// SIMATIC STEP 7 (V5.x) project S_M_General
// CPU: CPU312(1)
// station: P_ADR_BUS
// station: Hardware
// station: Equipo SIMATIC 300
// program: Programa S7(1)

SYMBOL_TABLE
"CONTADOR"	C 1	COUNTER
"Global"	DB 1	DB 1
"INFO_BOB"	DB 4	DB 4
"DESBOBINADO"	FB 1	FB 1	// Función que se encarga del desbobinado
"CIZALLADO"	FB 2	FB 2	// Funcion que se encaga del cizallado de planchas
"MULT_DESBOB"	FB 3	FB 3
"MULT_CIZA"	FB 4	FB 4
"MULT_GEN"	FB 5	FB 5
"MULT_GEN_DESB"	FB 6	FB 6
"CORTAR"	FC 1	FC 1	// Funcion de cortar las planchas
"PESAJE"	FC 2	FC 2	// Función de pesaje
"SCALE"	FC 105	FC 105	// Scaling Values
"START"	I 124.0	BOOL
"BIT_DE_TRABAJO"	I 124.1	BOOL
"BOBINA_COLOCADA"	I 124.2	BOOL
"S_SARTEN"	I 124.5	BOOL
"S_CACEROLA"	I 124.6	BOOL
"S_PAELLERA"	I 124.7	BOOL
"S_WOK"	I 125.0	BOOL
"PRESENCIA"	I 125.1	BOOL
"PALET"	I 125.3	BOOL
"SENSORARRIBA"	I 125.4	BOOL
"SENSORABAJO"	I 125.5	BOOL
"EXPULSADA"	I 125.6	BOOL
"PESO_OUT"	MD 100	REAL
"Cycle Execution"	OB 1	OB 1
"MCENTRO"	PIW 651	INT
"IN_PESAJE"	PIW 653	INT
"ABRIRMCENTRO"	Q 100.0	BOOL
"CERRARMCENTRO"	Q 100.1	BOOL
"DESBOBINAR"	Q 100.2	BOOL
"EXPULSAR_BOBINA"	Q 100.3	BOOL
"PRENSA"	Q 100.4	BOOL
"EXPULSAR_PLANCHA"	Q 100.5	BOOL
"BAJAR_CUCHILLA"	Q 100.6	BOOL
"EXPULSAR_PALET"	Q 101.0	BOOL
"STBY"	Q 101.1	BOOL
END_SYMBOL_TABLE

FUNCTION_BLOCK "DESBOBINADO"	// FB 1
TITLE = DESBOBINADO
VERSION : 0.1
VAR_INPUT
  SENSOR : BOOL ;
  PRESENCIA : BOOL ;
  CENTRO : INT ;
  bit_de_trabajo : BOOL ;
  MCENTRO : INT ;
  Contador : COUNTER ;
  START : BOOL ;
  PLANCHAS : WORD  := W#16#100;
END_VAR
VAR_OUTPUT
  ABRIRMCENTRO : BOOL ;
  DESBOBINAR : BOOL ;
  STBY : BOOL ;
END_VAR
VAR
  x31 : BOOL ;
  x32 : BOOL ;
  x33 : BOOL ;
  x34 : BOOL ;
  s1 : BOOL ;
  FP_Bit_Tr : BOOL ;
  x30 : BOOL ;
  FP_PRESENCIA : BOOL ;
  FP_BDT : BOOL ;
  FP_START : BOOL ;
END_VAR
VAR_TEMP
  watchdog_master : BOOL ;
END_VAR
BEGIN
NETWORK
TITLE = Arranque
      SET;
      A     #bit_de_trabajo;
      FP    #FP_BDT;
      S     #x30;
      R     #x31;
      R     #x32;
      R     #x33;
      R     #x34;
      R     #s1;
NETWORK
TITLE = x31 a x32
//Comparacion medida centro con medida nominal del centro para pasar de x31 a x32
      A     #x31;
      A(;
      L     #CENTRO;
      L     #MCENTRO;
      ==R;
      );
      R     #x31;
      S     #x32;
NETWORK
TITLE = x32 a x33
//Presencia detecta que la plancha esta en posicion para empezar el proceso de 
//desbobinado-cizallado
      A     #x32;
      A     #PRESENCIA;
      FP    #FP_PRESENCIA;
      R     #x32;
      S     #x33;
NETWORK
TITLE = x33 a x34
//Detecta que la plancha esta lista para ser cizallada
      A     #x33;
      A     #SENSOR;
      R     #x33;
      S     #x34;
NETWORK
TITLE = x34 a x33
//si el contador no ha acabado
      A     #x34;
      T     LD 1;
      TAK;
      T     LD 5;
      L     #Contador;
      T     LW 9;
      L     LD 5;
      L     LD 1;
      A     C [LW 9];
      AN    #SENSOR;
      R     #x34;
      S     #x33;
NETWORK
TITLE = x34 a s1
//si el contador ha cabado
      A     #x34;
      T     LD 1;
      TAK;
      T     LD 5;
      L     #Contador;
      T     LW 9;
      L     LD 5;
      L     LD 1;
      AN    C [LW 9];
      AN    #SENSOR;
      AN    #PRESENCIA;
      R     #x34;
      S     #x30;
NETWORK
TITLE = Tratamiento de bit de fin
      A     #x30;
      =     #STBY;
NETWORK
TITLE = Abrir centro
      A     #x31;
      =     #ABRIRMCENTRO;
NETWORK
TITLE = Carga del contador y desbobinado en x32
      A     #x32;
      S     #DESBOBINAR;
      L     #PLANCHAS;
      T     LD 1;
      TAK;
      T     LD 5;
      L     #Contador;
      T     LW 9;
      L     LD 5;
      L     LD 1;
      S     C [LW 9];
NETWORK
TITLE = Resta del contador y salida del x33
      A     #x33;
      S     #DESBOBINAR;
NETWORK
TITLE =
      A     #x34;
      R     #DESBOBINAR;
NETWORK
TITLE = De X30 a X31
      A     #START;
      FP    #FP_START;
      A     #x30;
      R     #x30;
      S     #x31;
END_FUNCTION_BLOCK

FUNCTION_BLOCK "CIZALLADO"	// FB 2
TITLE = CIZALLADO
VERSION : 0.1
VAR_INPUT
  bit_de_trabajo : BOOL ;
  SENSOR : BOOL ;
  SENSORABAJO : BOOL ;
  SENSORARRIBA : BOOL ;
  EXPULSADA : BOOL ;
  CONTADOR : COUNTER ;
  START : BOOL ;
END_VAR
VAR_OUTPUT
  BAJARCUCHILLA : BOOL ;
  EXPULSARPLANCHA : BOOL ;
  STBY : BOOL ;
  BIT_OK : BOOL ;
END_VAR
VAR
  X41 : BOOL ;
  M3 : BOOL ;
  X43 : BOOL ;
  FP_BDT : BOOL ;
  FP_START : BOOL ;
  INICORTAR : BOOL ;
  S2 : BOOL ;
  BDT_CORTAR : BOOL ;
  OK_CORTAR : BOOL ;
  STBY_CORTAR : BOOL ;
  CORTADO : BOOL ;
END_VAR
BEGIN
NETWORK
TITLE = Arranque
      A     #bit_de_trabajo;
      FP    #FP_BDT;
      =     #BDT_CORTAR;
      S     #X41;
      R     #M3;
      R     #X43;
      R     #INICORTAR;
      R     #CORTADO;
      R     #BIT_OK;
      R     #S2;
NETWORK
TITLE = De x41 a M3
      A     #X41;
      A     #SENSOR;
      A     #STBY_CORTAR;
      A     #START;
      FP    #FP_START;
      R     #X41;
      S     #M3;
NETWORK
TITLE = De M3 a x43
      A     #M3;
      A     #CORTADO;
      R     #M3;
      S     #X43;
NETWORK
TITLE = de x43 a x41
      A     #X43;
      T     LD 0;
      TAK;
      T     LD 4;
      L     #CONTADOR;
      T     LW 8;
      L     LD 4;
      L     LD 0;
      AN    C [LW 8];
      R     #X43;
      S     #S2;
NETWORK
TITLE = de x43 a X41
      A     #X43;
      T     LD 0;
      TAK;
      T     LD 4;
      L     #CONTADOR;
      T     LW 8;
      L     LD 4;
      L     LD 0;
      A     C [LW 8];
      R     #X43;
      S     #X41;
NETWORK
TITLE = De M3 a x43 con call M3
      CALL  "CORTAR" (
           bit_de_trabajo           := #BDT_CORTAR,
           SENSORABAJO              := #SENSORABAJO,
           SENSORARRIBA             := #SENSORARRIBA,
           EXPULSADA                := #EXPULSADA,
           START                    := #INICORTAR,
           OK                       := #OK_CORTAR,
           BAJARCUCHILLA            := #BAJARCUCHILLA,
           EXPULSARPLANCHA          := #EXPULSARPLANCHA,
           bit_ok                   := #CORTADO,
           STBY                     := #STBY_CORTAR);
NETWORK
TITLE =
      A     #M3;
      A     #CORTADO;
      R     #M3;
      S     #X43;
NETWORK
TITLE =
      A     #M3;
      =     #INICORTAR;
NETWORK
TITLE = Cuenta el numero de planchas cortadas
      A     #X43;
      =     #OK_CORTAR;
      T     LD 0;
      TAK;
      T     LD 4;
      L     #CONTADOR;
      T     LW 8;
      L     LD 4;
      L     LD 0;
      CD    C [LW 8];
NETWORK
TITLE =
      A     #X41;
      =     #STBY;
NETWORK
TITLE =
      A     #S2;
      =     #BIT_OK;
END_FUNCTION_BLOCK

FUNCTION_BLOCK "MULT_DESBOB"	// FB 3
VERSION : 0.1
VAR_INPUT
  S_CACEROLA : BOOL ;
  S_SARTEN : BOOL ;
  S_PAELLERA : BOOL ;
  S_WOK : BOOL ;
  PRESENCIA : BOOL ;
  C_CACEROLA : INT ;
  C_SARTEN : INT ;
  C_WOK : INT ;
  C_PAELLERA : INT ;
  BIT_DE_TRABAJO : BOOL ;
  MCENTRO : INT ;
  CONTADOR : COUNTER ;
  PLANCHAS : WORD ;
  SARTEN : BOOL ;
  CACEROLA : BOOL ;
  WOK : BOOL ;
  PAELLERA : BOOL ;
  START : BOOL ;
END_VAR
VAR_OUTPUT
  ABRIRMCENTRO : BOOL ;
  DESBOBINAR : BOOL ;
  BIT_OK : BOOL ;
  BIT_ERROR : BOOL ;
  STBY : BOOL ;
END_VAR
VAR
  CAC_DESB : FB 1;
  SART_DESB : FB 1;
  WOK_DESB : FB 1;
  PAELL_DESB : FB 1;
  START_SAR : BOOL ;
  START_CAC : BOOL ;
  START_WOK : BOOL ;
  START_PAELL : BOOL ;
  FP_BDT : BOOL ;
  X1 : BOOL ;
  X2 : BOOL ;
  X3 : BOOL ;
  X4 : BOOL ;
  X5 : BOOL ;
  X6 : BOOL ;
  BDT : BOOL ;
  FP_START : BOOL ;
  FLAG_DESB : BOOL ;
  FP_DESBOB : BOOL ;
  F_START : BOOL ;
  STBY_SAR : BOOL ;
  STBY_CAC : BOOL ;
  STBY_WOK : BOOL ;
  STBY_PAELL : BOOL ;
END_VAR
BEGIN
NETWORK
TITLE =
      A     #X2;
      JCN   _008;
      S     #BDT;
      BLD   14;
      =     L 6.0;
      L     DINO;
      T     LW 4;
      CDB;
      OPN   DI [LW 4];
      TAR2  LD 0;
      A     DBX [AR2,P#0.1];
      =     #SART_DESB.SENSOR;
      A     DBX [AR2,P#0.4];
      =     #SART_DESB.PRESENCIA;
      L     DBW [AR2,P#4.0];
      T     #SART_DESB.CENTRO;
      A     DBX [AR2,P#95.3];
      =     #SART_DESB.bit_de_trabajo;
      L     DBW [AR2,P#12.0];
      T     #SART_DESB.MCENTRO;
      L     DBW [AR2,P#14.0];
      T     #SART_DESB.Contador;
      A     DBX [AR2,P#94.0];
      =     #SART_DESB.START;
      L     DBW [AR2,P#16.0];
      T     #SART_DESB.PLANCHAS;
      +AR2  P#40.0;
      UC    "DESBOBINADO";
      LAR2  LD 0;
      A     #SART_DESB.ABRIRMCENTRO;
      =     DBX [AR2,P#20.0];
      A     #SART_DESB.DESBOBINAR;
      =     DBX [AR2,P#20.1];
      A     #SART_DESB.STBY;
      =     DBX [AR2,P#96.0];
      CDB;
      BLD   15;
_008: NOP   0;
NETWORK
TITLE =
      A     #X3;
      JCN   _009;
      S     #BDT;
      BLD   14;
      =     L 6.0;
      L     DINO;
      T     LW 4;
      CDB;
      OPN   DI [LW 4];
      TAR2  LD 0;
      A     DBX [AR2,P#0.0];
      =     #CAC_DESB.SENSOR;
      A     DBX [AR2,P#0.4];
      =     #CAC_DESB.PRESENCIA;
      L     DBW [AR2,P#2.0];
      T     #CAC_DESB.CENTRO;
      A     DBX [AR2,P#95.3];
      =     #CAC_DESB.bit_de_trabajo;
      L     DBW [AR2,P#12.0];
      T     #CAC_DESB.MCENTRO;
      L     DBW [AR2,P#14.0];
      T     #CAC_DESB.Contador;
      A     DBX [AR2,P#94.1];
      =     #CAC_DESB.START;
      L     DBW [AR2,P#16.0];
      T     #CAC_DESB.PLANCHAS;
      +AR2  P#22.0;
      UC    "DESBOBINADO";
      LAR2  LD 0;
      A     #CAC_DESB.ABRIRMCENTRO;
      =     DBX [AR2,P#20.0];
      A     #CAC_DESB.DESBOBINAR;
      =     DBX [AR2,P#20.1];
      A     #CAC_DESB.STBY;
      =     DBX [AR2,P#96.1];
      CDB;
      BLD   15;
_009: NOP   0;
NETWORK
TITLE =
      A     #X4;
      JCN   _010;
      S     #BDT;
      BLD   14;
      =     L 6.0;
      L     DINO;
      T     LW 4;
      CDB;
      OPN   DI [LW 4];
      TAR2  LD 0;
      A     DBX [AR2,P#0.3];
      =     #WOK_DESB.SENSOR;
      A     DBX [AR2,P#0.4];
      =     #WOK_DESB.PRESENCIA;
      L     DBW [AR2,P#6.0];
      T     #WOK_DESB.CENTRO;
      A     DBX [AR2,P#95.3];
      =     #WOK_DESB.bit_de_trabajo;
      L     DBW [AR2,P#12.0];
      T     #WOK_DESB.MCENTRO;
      L     DBW [AR2,P#14.0];
      T     #WOK_DESB.Contador;
      A     DBX [AR2,P#94.2];
      =     #WOK_DESB.START;
      L     DBW [AR2,P#16.0];
      T     #WOK_DESB.PLANCHAS;
      +AR2  P#58.0;
      UC    "DESBOBINADO";
      LAR2  LD 0;
      A     #WOK_DESB.ABRIRMCENTRO;
      =     DBX [AR2,P#20.0];
      A     #WOK_DESB.DESBOBINAR;
      =     DBX [AR2,P#20.1];
      A     #WOK_DESB.STBY;
      =     DBX [AR2,P#96.2];
      CDB;
      BLD   15;
_010: NOP   0;
NETWORK
TITLE =
      A     #X5;
      JCN   _011;
      S     #BDT;
      BLD   14;
      =     L 6.0;
      L     DINO;
      T     LW 4;
      CDB;
      OPN   DI [LW 4];
      TAR2  LD 0;
      A     DBX [AR2,P#0.2];
      =     #PAELL_DESB.SENSOR;
      A     DBX [AR2,P#0.4];
      =     #PAELL_DESB.PRESENCIA;
      L     DBW [AR2,P#8.0];
      T     #PAELL_DESB.CENTRO;
      A     DBX [AR2,P#95.3];
      =     #PAELL_DESB.bit_de_trabajo;
      L     DBW [AR2,P#12.0];
      T     #PAELL_DESB.MCENTRO;
      L     DBW [AR2,P#14.0];
      T     #PAELL_DESB.Contador;
      A     DBX [AR2,P#94.3];
      =     #PAELL_DESB.START;
      L     DBW [AR2,P#16.0];
      T     #PAELL_DESB.PLANCHAS;
      +AR2  P#76.0;
      UC    "DESBOBINADO";
      LAR2  LD 0;
      A     #PAELL_DESB.ABRIRMCENTRO;
      =     DBX [AR2,P#20.0];
      A     #PAELL_DESB.DESBOBINAR;
      =     DBX [AR2,P#20.1];
      A     #PAELL_DESB.STBY;
      =     DBX [AR2,P#96.3];
      CDB;
      BLD   15;
_011: NOP   0;
NETWORK
TITLE =
      A     #X2;
      =     #START_SAR;
NETWORK
TITLE =
      A     #X3;
      =     #START_CAC;
NETWORK
TITLE =
      A     #X4;
      =     #START_WOK;
NETWORK
TITLE =
      A     #X5;
      =     #START_PAELL;
NETWORK
TITLE =
      A     #BIT_DE_TRABAJO;
      FP    #FP_BDT;
      R     #START_SAR;
      R     #START_CAC;
      R     #START_WOK;
      R     #START_PAELL;
      S     #X1;
      R     #X2;
      R     #X3;
      R     #X4;
      R     #X5;
      R     #X6;
NETWORK
TITLE =
      A     #START;
      FP    #FP_START;
      =     #F_START;
NETWORK
TITLE =
      A     #F_START;
      A     #X1;
      A     #SARTEN;
      R     #X1;
      S     #X2;
NETWORK
TITLE =
      A     #F_START;
      A     #X1;
      A     #CACEROLA;
      R     #X1;
      S     #X3;
NETWORK
TITLE =
      A     #F_START;
      A     #X1;
      A     #WOK;
      R     #X1;
      S     #X4;
NETWORK
TITLE =
      A     #F_START;
      A     #X1;
      A     #PAELLERA;
      R     #X1;
      S     #X5;
NETWORK
TITLE =
      A     #DESBOBINAR;
      FP    #FP_DESBOB;
      S     #FLAG_DESB;
NETWORK
TITLE =
      A     #X2;
      A     #FLAG_DESB;
      A     #STBY_SAR;
      R     #FLAG_DESB;
      R     #X2;
      S     #X6;
NETWORK
TITLE =
      A     #X3;
      A     #FLAG_DESB;
      A     #STBY_CAC;
      R     #FLAG_DESB;
      R     #X3;
      S     #X6;
NETWORK
TITLE =
      A     #X4;
      A     #FLAG_DESB;
      A     #STBY_WOK;
      R     #FLAG_DESB;
      R     #X4;
      S     #X6;
NETWORK
TITLE =
      A     #X5;
      A     #FLAG_DESB;
      A     #STBY_PAELL;
      R     #FLAG_DESB;
      R     #X5;
      S     #X6;
NETWORK
TITLE =
      A     #X1;
      =     #STBY;
NETWORK
TITLE =
      A     #X6;
      =     #BIT_OK;
END_FUNCTION_BLOCK

FUNCTION_BLOCK "MULT_CIZA"	// FB 4
VERSION : 0.1
VAR_INPUT
  S_CACEROLA : BOOL ;
  S_WOK : BOOL ;
  S_SARTEN : BOOL ;
  S_PAELLERA : BOOL ;
  BIT_DE_TRABAJO : BOOL ;
  SENSORARRIBA : BOOL ;
  SENSORABAJO : BOOL ;
  EXPULSADA : BOOL ;
  CONTADOR : COUNTER ;
  SARTEN : BOOL ;
  CACEROLA : BOOL ;
  WOK : BOOL ;
  PAELLERA : BOOL ;
  START : BOOL ;
END_VAR
VAR_OUTPUT
  EXPULSARPLANCHA : BOOL ;
  BAJARCUCHILLA : BOOL ;
  BIT_OK : BOOL ;
  STBY : BOOL ;
END_VAR
VAR
  BDT : BOOL ;
  START_SAR : BOOL ;
  START_CAC : BOOL ;
  START_WOK : BOOL ;
  START_PAELL : BOOL ;
  X1 : BOOL ;
  X2 : BOOL ;
  X3 : BOOL ;
  X4 : BOOL ;
  X5 : BOOL ;
  FP_START : BOOL ;
  F_START : BOOL ;
  STBY_SAR : BOOL ;
  STBY_CAC : BOOL ;
  STBY_WOK : BOOL ;
  STBY_PAELL : BOOL ;
  OK : BOOL ;
  FP_BDT : BOOL ;
  CAC_CIZA : FB 2;
  SART_CIZA : FB 2;
  WOK_CIZA : FB 2;
  PAELL_CIZA : FB 2;
  X6 : BOOL ;
END_VAR
BEGIN
NETWORK
TITLE =
      A     #BIT_DE_TRABAJO;
      FP    #FP_BDT;
      S     #X1;
      R     #X2;
      R     #X3;
      R     #X4;
      R     #X5;
      R     #X6;
NETWORK
TITLE =
      A     #START;
      FP    #FP_START;
      =     #F_START;
NETWORK
TITLE =
      A     #F_START;
      A     #SARTEN;
      A     #X1;
      R     #X1;
      S     #X2;
NETWORK
TITLE =
      A     #F_START;
      A     #CACEROLA;
      A     #X1;
      R     #X1;
      S     #X3;
NETWORK
TITLE =
      A     #F_START;
      A     #WOK;
      A     #X1;
      R     #X1;
      S     #X4;
NETWORK
TITLE =
      A     #F_START;
      A     #PAELLERA;
      A     #X1;
      R     #X1;
      S     #X5;
NETWORK
TITLE =
      A     #OK;
      A(;
      O     #X2;
      O     #X3;
      O     #X4;
      O     #X5;
      );
      R     #X2;
      R     #X3;
      R     #X4;
      R     #X5;
      S     #X6;
NETWORK
TITLE =
      A     #X2;
      JCN   _001;
      S     #BDT;
      BLD   14;
      =     L 6.0;
      L     DINO;
      T     LW 4;
      CDB;
      OPN   DI [LW 4];
      TAR2  LD 0;
      A     DBX [AR2,P#8.0];
      =     #SART_CIZA.bit_de_trabajo;
      A     DBX [AR2,P#0.2];
      =     #SART_CIZA.SENSOR;
      A     DBX [AR2,P#0.6];
      =     #SART_CIZA.SENSORABAJO;
      A     DBX [AR2,P#0.5];
      =     #SART_CIZA.SENSORARRIBA;
      A     DBX [AR2,P#0.7];
      =     #SART_CIZA.EXPULSADA;
      L     DBW [AR2,P#2.0];
      T     #SART_CIZA.CONTADOR;
      A     DBX [AR2,P#4.4];
      =     #SART_CIZA.START;
      +AR2  P#22.0;
      UC    "CIZALLADO";
      LAR2  LD 0;
      A     #SART_CIZA.BAJARCUCHILLA;
      =     DBX [AR2,P#6.1];
      A     #SART_CIZA.EXPULSARPLANCHA;
      =     DBX [AR2,P#6.0];
      A     #SART_CIZA.STBY;
      =     DBX [AR2,P#6.3];
      A     #SART_CIZA.BIT_OK;
      =     DBX [AR2,P#10.0];
      CDB;
      BLD   15;
_001: NOP   0;
NETWORK
TITLE =
      A     #X3;
      JCN   _002;
      S     #BDT;
      BLD   14;
      =     L 6.0;
      L     DINO;
      T     LW 4;
      CDB;
      OPN   DI [LW 4];
      TAR2  LD 0;
      A     DBX [AR2,P#8.0];
      =     #CAC_CIZA.bit_de_trabajo;
      A     DBX [AR2,P#0.0];
      =     #CAC_CIZA.SENSOR;
      A     DBX [AR2,P#0.6];
      =     #CAC_CIZA.SENSORABAJO;
      A     DBX [AR2,P#0.5];
      =     #CAC_CIZA.SENSORARRIBA;
      A     DBX [AR2,P#0.7];
      =     #CAC_CIZA.EXPULSADA;
      L     DBW [AR2,P#2.0];
      T     #CAC_CIZA.CONTADOR;
      A     DBX [AR2,P#4.4];
      =     #CAC_CIZA.START;
      +AR2  P#12.0;
      UC    "CIZALLADO";
      LAR2  LD 0;
      A     #CAC_CIZA.BAJARCUCHILLA;
      =     DBX [AR2,P#6.1];
      A     #CAC_CIZA.EXPULSARPLANCHA;
      =     DBX [AR2,P#6.0];
      A     #CAC_CIZA.STBY;
      =     DBX [AR2,P#6.3];
      A     #CAC_CIZA.BIT_OK;
      =     DBX [AR2,P#10.0];
      CDB;
      BLD   15;
_002: NOP   0;
NETWORK
TITLE =
      A     #X4;
      JCN   _003;
      S     #BDT;
      BLD   14;
      =     L 6.0;
      L     DINO;
      T     LW 4;
      CDB;
      OPN   DI [LW 4];
      TAR2  LD 0;
      A     DBX [AR2,P#8.0];
      =     #WOK_CIZA.bit_de_trabajo;
      A     DBX [AR2,P#0.1];
      =     #WOK_CIZA.SENSOR;
      A     DBX [AR2,P#0.6];
      =     #WOK_CIZA.SENSORABAJO;
      A     DBX [AR2,P#0.5];
      =     #WOK_CIZA.SENSORARRIBA;
      A     DBX [AR2,P#0.7];
      =     #WOK_CIZA.EXPULSADA;
      L     DBW [AR2,P#2.0];
      T     #WOK_CIZA.CONTADOR;
      A     DBX [AR2,P#4.4];
      =     #WOK_CIZA.START;
      +AR2  P#32.0;
      UC    "CIZALLADO";
      LAR2  LD 0;
      A     #WOK_CIZA.BAJARCUCHILLA;
      =     DBX [AR2,P#6.1];
      A     #WOK_CIZA.EXPULSARPLANCHA;
      =     DBX [AR2,P#6.0];
      A     #WOK_CIZA.STBY;
      =     DBX [AR2,P#6.3];
      A     #WOK_CIZA.BIT_OK;
      =     DBX [AR2,P#10.0];
      CDB;
      BLD   15;
_003: NOP   0;
NETWORK
TITLE =
      A     #X5;
      JCN   _004;
      S     #BDT;
      BLD   14;
      =     L 6.0;
      L     DINO;
      T     LW 4;
      CDB;
      OPN   DI [LW 4];
      TAR2  LD 0;
      A     DBX [AR2,P#8.0];
      =     #PAELL_CIZA.bit_de_trabajo;
      A     DBX [AR2,P#0.3];
      =     #PAELL_CIZA.SENSOR;
      A     DBX [AR2,P#0.6];
      =     #PAELL_CIZA.SENSORABAJO;
      A     DBX [AR2,P#0.5];
      =     #PAELL_CIZA.SENSORARRIBA;
      A     DBX [AR2,P#0.7];
      =     #PAELL_CIZA.EXPULSADA;
      L     DBW [AR2,P#2.0];
      T     #PAELL_CIZA.CONTADOR;
      A     DBX [AR2,P#4.4];
      =     #PAELL_CIZA.START;
      +AR2  P#42.0;
      UC    "CIZALLADO";
      LAR2  LD 0;
      A     #PAELL_CIZA.BAJARCUCHILLA;
      =     DBX [AR2,P#6.1];
      A     #PAELL_CIZA.EXPULSARPLANCHA;
      =     DBX [AR2,P#6.0];
      A     #PAELL_CIZA.STBY;
      =     DBX [AR2,P#6.3];
      A     #PAELL_CIZA.BIT_OK;
      =     DBX [AR2,P#10.0];
      CDB;
      BLD   15;
_004: NOP   0;
NETWORK
TITLE =
      A     #X2;
      =     #START_SAR;
NETWORK
TITLE =
      A     #X3;
      =     #START_CAC;
NETWORK
TITLE =
      A     #X4;
      =     #START_WOK;
NETWORK
TITLE =
      A     #X5;
      =     #START_PAELL;
NETWORK
TITLE =
      A     #X1;
      =     #STBY;
NETWORK
TITLE =
      A     #X6;
      =     #BIT_OK;
      R     #BDT;
      R     #OK;
END_FUNCTION_BLOCK

FUNCTION_BLOCK "MULT_GEN"	// FB 5
VERSION : 0.1
VAR_INPUT
  START : BOOL ;
  BIT_DE_TRABAJO : BOOL ;
  BOBINA_COLOCADA : BOOL ;
  MCENTRO : INT ;
  IN_PESAJE : INT ;
  S_SARTEN : BOOL ;
  S_CACEROLA : BOOL ;
  S_WOK : BOOL ;
  S_PAELLERA : BOOL ;
  PRESENCIA : BOOL ;
  CONTADOR : COUNTER ;
  PALET : BOOL ;
  SENSORARRIBA : BOOL ;
  SENSORABAJO : BOOL ;
  EXPULSADA : BOOL ;
END_VAR
VAR_OUTPUT
  PESO_OUT : REAL ;
  ABRIRMCENTRO : BOOL ;
  CERRARMCENTRO : BOOL ;
  DESBOBINAR : BOOL ;
  EXPULSAR_BOBINA : BOOL ;
  PRENSA : BOOL ;
  EXPULSAR_PLANCHA : BOOL ;
  BAJAR_CUCHILLA : BOOL ;
  EXPULSAR_PALET : BOOL ;
  STBY : BOOL ;
END_VAR
VAR
  X0 : BOOL ;
  X1 : BOOL ;
  X2 : BOOL ;
  X3 : BOOL ;
  X4 : BOOL ;
  X5 : BOOL ;
  FP_START : BOOL ;
  BDT_PESAJE : BOOL ;
  RECIBIDO_PESAJE : BOOL ;
  START_PESAJE : BOOL ;
  STBY_PESAJE : BOOL ;
  SARTEN : BOOL ;
  CACEROLA : BOOL ;
  WOK : BOOL ;
  PAELLERA : BOOL ;
  OK_DESBOB : BOOL ;
  DESBOB : FB 3;
  BDT_DESBOB : BOOL ;
  START_DESBOB : BOOL ;
  OK_DESBOB_1 : BOOL ;
  STBY_DESBOB : BOOL ;
  X10 : BOOL ;
  X11 : BOOL ;
  X12 : BOOL ;
  FP_BDT : BOOL ;
  OK_CIZA : BOOL ;
  CIZA : FB 4;
  BDT_CIZA : BOOL ;
  START_CIZA : BOOL ;
  STBY_CIZA : BOOL ;
  FP_OK_DESBOB : BOOL ;
  FP_OK_CIZA : BOOL ;
END_VAR
BEGIN
NETWORK
TITLE =
      A     #BIT_DE_TRABAJO;
      FP    #FP_BDT;
      S     #X0;
      R     #X1;
      R     #X2;
      R     #X3;
      R     #X4;
      R     #X5;
      R     #X10;
      R     #X11;
      R     #X12;
      R     #OK_DESBOB;
      R     #OK_CIZA;
NETWORK
TITLE =
      A     #START;
      FP    #FP_START;
      A     #X0;
      R     #X0;
      S     #X1;
      S     #X10;
NETWORK
TITLE =
      A     #X1;
      A     #BOBINA_COLOCADA;
      R     #X1;
      S     #X2;
NETWORK
TITLE =
      A     #X2;
      A(;
      O     #SARTEN;
      O     #CACEROLA;
      O     #WOK;
      O     #PAELLERA;
      );
      R     #X2;
      S     #X3;
NETWORK
TITLE =
      A     #OK_DESBOB;
      FP    #FP_OK_DESBOB;
      A     #X3;
      R     #X3;
      R     #OK_DESBOB;
      S     #X4;
NETWORK
TITLE =
      A     #X4;
      A(;
      L     #MCENTRO;
      L     0;
      ==I;
      );
      R     #X4;
      S     #X5;
NETWORK
TITLE =
      A     #X2;
      JCN   _001;
      S     #BDT_PESAJE;
      CALL  "PESAJE" (
           in                       := #IN_PESAJE,
           PESO_SARTEN              := "Global".PESO_SARTEN,
           PESO_CACEROLA            := "Global".PESO_CACEROLA,
           PESO_WOK                 := "Global".PESO_WOK,
           PESO_PAELLERA            := "Global".PESO_PAELLERA,
           bit_de_trabajo           := #BDT_PESAJE,
           RECIBIDO                 := #RECIBIDO_PESAJE,
           START                    := #START_PESAJE,
           stby                     := #STBY_PESAJE,
           SARTEN                   := #SARTEN,
           CACEROLA                 := #CACEROLA,
           WOK                      := #WOK,
           PAELLERA                 := #PAELLERA,
           PESO_OUT                 := #PESO_OUT);
_001: NOP   0;
NETWORK
TITLE =
      A     #X2;
      =     #START_PESAJE;
NETWORK
TITLE =
      A     #X3;
      =     #START_DESBOB;
NETWORK
TITLE =
      A     #X4;
      =     #CERRARMCENTRO;
      R     #BDT_DESBOB;
NETWORK
TITLE =
      A     #X5;
      =     #EXPULSAR_BOBINA;
NETWORK
TITLE =
      A     #DESBOBINAR;
      =     #PRENSA;
NETWORK
TITLE =
      A     #X10;
      A(;
      O     #SARTEN;
      O     #CACEROLA;
      O     #WOK;
      O     #PAELLERA;
      );
      R     #X10;
      S     #X11;
NETWORK
TITLE =
      A     #OK_CIZA;
      FP    #FP_OK_CIZA;
      A     #X11;
      R     #X11;
      S     #X12;
NETWORK
TITLE =
      A     #X11;
      JCN   _003;
      S     #BDT_CIZA;
      BLD   14;
      =     L 6.0;
      L     DINO;
      T     LW 4;
      CDB;
      OPN   DI [LW 4];
      TAR2  LD 0;
      A     DBX [AR2,P#6.1];
      =     #CIZA.S_CACEROLA;
      A     DBX [AR2,P#6.2];
      =     #CIZA.S_WOK;
      A     DBX [AR2,P#6.0];
      =     #CIZA.S_SARTEN;
      A     DBX [AR2,P#6.3];
      =     #CIZA.S_PAELLERA;
      A     DBX [AR2,P#174.0];
      =     #CIZA.BIT_DE_TRABAJO;
      A     DBX [AR2,P#10.1];
      =     #CIZA.SENSORARRIBA;
      A     DBX [AR2,P#10.2];
      =     #CIZA.SENSORABAJO;
      A     DBX [AR2,P#10.3];
      =     #CIZA.EXPULSADA;
      L     DBW [AR2,P#8.0];
      T     #CIZA.CONTADOR;
      A     DBX [AR2,P#19.3];
      =     #CIZA.SARTEN;
      A     DBX [AR2,P#19.4];
      =     #CIZA.CACEROLA;
      A     DBX [AR2,P#19.5];
      =     #CIZA.WOK;
      A     DBX [AR2,P#19.6];
      =     #CIZA.PAELLERA;
      A     DBX [AR2,P#174.1];
      =     #CIZA.START;
      +AR2  P#120.0;
      UC    "MULT_CIZA";
      LAR2  LD 0;
      A     #CIZA.EXPULSARPLANCHA;
      =     DBX [AR2,P#16.5];
      A     #CIZA.BAJARCUCHILLA;
      =     DBX [AR2,P#16.6];
      A     #CIZA.BIT_OK;
      =     DBX [AR2,P#119.0];
      A     #CIZA.STBY;
      =     DBX [AR2,P#174.2];
      CDB;
      BLD   15;
_003: NOP   0;
NETWORK
TITLE =
      A     #X11;
      =     #START_CIZA;
NETWORK
TITLE =
      A     #X3;
      JCN   _002;
      S     #BDT_DESBOB;
      R     #BDT_PESAJE;
      BLD   14;
      =     L 6.0;
      L     DINO;
      T     LW 4;
      CDB;
      OPN   DI [LW 4];
      TAR2  LD 0;
      A     DBX [AR2,P#6.1];
      =     #DESBOB.S_CACEROLA;
      A     DBX [AR2,P#6.0];
      =     #DESBOB.S_SARTEN;
      A     DBX [AR2,P#6.3];
      =     #DESBOB.S_PAELLERA;
      A     DBX [AR2,P#6.2];
      =     #DESBOB.S_WOK;
      A     DBX [AR2,P#6.4];
      =     #DESBOB.PRESENCIA;
      OPN   DI 4;
      L     DIW 0;
      OPN   DI [LW 4];
      T     #DESBOB.C_CACEROLA;
      OPN   DI 4;
      L     DIW 2;
      OPN   DI [LW 4];
      T     #DESBOB.C_SARTEN;
      OPN   DI 4;
      L     DIW 4;
      OPN   DI [LW 4];
      T     #DESBOB.C_WOK;
      OPN   DI 4;
      L     DIW 6;
      OPN   DI [LW 4];
      T     #DESBOB.C_PAELLERA;
      A     DBX [AR2,P#118.0];
      =     #DESBOB.BIT_DE_TRABAJO;
      L     DBW [AR2,P#2.0];
      T     #DESBOB.MCENTRO;
      L     DBW [AR2,P#8.0];
      T     #DESBOB.CONTADOR;
      OPN   DI 1;
      L     DIW 16;
      OPN   DI [LW 4];
      T     #DESBOB.PLANCHAS;
      A     DBX [AR2,P#19.3];
      =     #DESBOB.SARTEN;
      A     DBX [AR2,P#19.4];
      =     #DESBOB.CACEROLA;
      A     DBX [AR2,P#19.5];
      =     #DESBOB.WOK;
      A     DBX [AR2,P#19.6];
      =     #DESBOB.PAELLERA;
      A     DBX [AR2,P#118.1];
      =     #DESBOB.START;
      +AR2  P#20.0;
      UC    "MULT_DESBOB";
      LAR2  LD 0;
      A     #DESBOB.ABRIRMCENTRO;
      =     DBX [AR2,P#16.0];
      A     #DESBOB.DESBOBINAR;
      =     DBX [AR2,P#16.2];
      A     #DESBOB.BIT_OK;
      =     DBX [AR2,P#19.7];
      A     #DESBOB.STBY;
      =     DBX [AR2,P#118.3];
      CDB;
      BLD   15;
_002: NOP   0;
NETWORK
TITLE =
      A     #X12;
      =     #EXPULSAR_PALET;
NETWORK
TITLE =
      A     #X5;
      A     #X12;
      A     #START;
      R     #X5;
      R     #X12;
      S     #X1;
      S     #X10;
NETWORK
TITLE =
      A     #X5;
      A     #X12;
      AN    #START;
      R     #X5;
      R     #X12;
      S     #X0;
NETWORK
TITLE =
      A     #X0;
      =     #STBY;
END_FUNCTION_BLOCK

FUNCTION_BLOCK "MULT_GEN_DESB"	// FB 6
VERSION : 0.1
VAR_INPUT
  START : BOOL ;
  BIT_DE_TRABAJO : BOOL ;
  BOBINA_COLOCADA : BOOL ;
  MCENTRO : INT ;
  IN_PESAJE : INT ;
  S_SARTEN : BOOL ;
  S_CACEROLA : BOOL ;
  S_WOK : BOOL ;
  S_PAELLERA : BOOL ;
  PRESENCIA : BOOL ;
  CONTADOR : COUNTER ;
END_VAR
VAR_OUTPUT
  PESO_OUT : REAL ;
  ABRIRMCENTRO : BOOL ;
  CERRARMCENTRO : BOOL ;
  DESBOBINAR : BOOL ;
  EXPULSAR_BOBINA : BOOL ;
END_VAR
VAR
  X0 : BOOL ;
  X1 : BOOL ;
  X2 : BOOL ;
  X3 : BOOL ;
  X4 : BOOL ;
  X5 : BOOL ;
  FP_START : BOOL ;
  BDT_PESAJE : BOOL ;
  RECIBIDO_PESAJE : BOOL ;
  START_PESAJE : BOOL ;
  STBY_PESAJE : BOOL ;
  SARTEN : BOOL ;
  CACEROLA : BOOL ;
  WOK : BOOL ;
  PAELLERA : BOOL ;
  OK_DESBOB : BOOL ;
  DESBOB : FB 3;
  BDT_DESBOB : BOOL ;
  START_DESBOB : BOOL ;
  OK_DESBOB_1 : BOOL ;
  STBY_DESBOB : BOOL ;
  FP_OK_DESBOB : BOOL ;
  FP_BDT : BOOL ;
END_VAR
BEGIN
NETWORK
TITLE =
      A     #X1;
      A     #BOBINA_COLOCADA;
      R     #X1;
      S     #X2;
NETWORK
TITLE =
      A     #START;
      FP    #FP_START;
      A     #X0;
      R     #X0;
      S     #X1;
NETWORK
TITLE =
      A     #BIT_DE_TRABAJO;
      FP    #FP_BDT;
      S     #X0;
      R     #X1;
      R     #X2;
      R     #X3;
      R     #X4;
      R     #X5;
      R     #OK_DESBOB;
NETWORK
TITLE =
      A     #X3;
      JCN   _002;
      S     #BDT_DESBOB;
      R     #BDT_PESAJE;
      BLD   14;
      =     L 6.0;
      L     DINO;
      T     LW 4;
      CDB;
      OPN   DI [LW 4];
      TAR2  LD 0;
      A     DBX [AR2,P#6.1];
      =     #DESBOB.S_CACEROLA;
      A     DBX [AR2,P#6.0];
      =     #DESBOB.S_SARTEN;
      A     DBX [AR2,P#6.3];
      =     #DESBOB.S_PAELLERA;
      A     DBX [AR2,P#6.2];
      =     #DESBOB.S_WOK;
      A     DBX [AR2,P#6.4];
      =     #DESBOB.PRESENCIA;
      OPN   DI 4;
      L     DIW 0;
      OPN   DI [LW 4];
      T     #DESBOB.C_CACEROLA;
      OPN   DI 4;
      L     DIW 2;
      OPN   DI [LW 4];
      T     #DESBOB.C_SARTEN;
      OPN   DI 4;
      L     DIW 4;
      OPN   DI [LW 4];
      T     #DESBOB.C_WOK;
      OPN   DI 4;
      L     DIW 6;
      OPN   DI [LW 4];
      T     #DESBOB.C_PAELLERA;
      A     DBX [AR2,P#116.0];
      =     #DESBOB.BIT_DE_TRABAJO;
      L     DBW [AR2,P#2.0];
      T     #DESBOB.MCENTRO;
      L     DBW [AR2,P#8.0];
      T     #DESBOB.CONTADOR;
      OPN   DI 1;
      L     DIW 16;
      OPN   DI [LW 4];
      T     #DESBOB.PLANCHAS;
      A     DBX [AR2,P#17.3];
      =     #DESBOB.SARTEN;
      A     DBX [AR2,P#17.4];
      =     #DESBOB.CACEROLA;
      A     DBX [AR2,P#17.5];
      =     #DESBOB.WOK;
      A     DBX [AR2,P#17.6];
      =     #DESBOB.PAELLERA;
      A     DBX [AR2,P#116.1];
      =     #DESBOB.START;
      +AR2  P#18.0;
      UC    "MULT_DESBOB";
      LAR2  LD 0;
      A     #DESBOB.ABRIRMCENTRO;
      =     DBX [AR2,P#14.0];
      A     #DESBOB.DESBOBINAR;
      =     DBX [AR2,P#14.2];
      A     #DESBOB.BIT_OK;
      =     DBX [AR2,P#17.7];
      A     #DESBOB.STBY;
      =     DBX [AR2,P#116.3];
      CDB;
      BLD   15;
_002: NOP   0;
NETWORK
TITLE =
      A     #X2;
      A(;
      O     #SARTEN;
      O     #CACEROLA;
      O     #WOK;
      O     #PAELLERA;
      );
      R     #X2;
      S     #X3;
NETWORK
TITLE =
      A     #OK_DESBOB;
      FP    #FP_OK_DESBOB;
      A     #X3;
      R     #X3;
      R     #OK_DESBOB;
      S     #X4;
NETWORK
TITLE =
      A     #X4;
      A(;
      L     #MCENTRO;
      L     0;
      ==I;
      );
      R     #X4;
      S     #X5;
NETWORK
TITLE =
      A     #X2;
      JCN   _001;
      S     #BDT_PESAJE;
      CALL  "PESAJE" (
           in                       := #IN_PESAJE,
           PESO_SARTEN              := "Global".PESO_SARTEN,
           PESO_CACEROLA            := "Global".PESO_CACEROLA,
           PESO_WOK                 := "Global".PESO_WOK,
           PESO_PAELLERA            := "Global".PESO_PAELLERA,
           bit_de_trabajo           := #BDT_PESAJE,
           RECIBIDO                 := #RECIBIDO_PESAJE,
           START                    := #START_PESAJE,
           stby                     := #STBY_PESAJE,
           SARTEN                   := #SARTEN,
           CACEROLA                 := #CACEROLA,
           WOK                      := #WOK,
           PAELLERA                 := #PAELLERA,
           PESO_OUT                 := #PESO_OUT);
_001: NOP   0;
NETWORK
TITLE =
      A     #X2;
      =     #START_PESAJE;
NETWORK
TITLE =
      A     #X3;
      =     #START_DESBOB;
NETWORK
TITLE =
      A     #X4;
      =     #CERRARMCENTRO;
      R     #BDT_DESBOB;
NETWORK
TITLE =
      A     #X5;
      =     #EXPULSAR_BOBINA;
END_FUNCTION_BLOCK

FUNCTION "CORTAR" : VOID	// FC 1
TITLE = CORTAR
VERSION : 0.1
VAR_INPUT
  bit_de_trabajo : BOOL ;
  SENSORABAJO : BOOL ;
  SENSORARRIBA : BOOL ;
  EXPULSADA : BOOL ;
  START : BOOL ;
  OK : BOOL ;
END_VAR
VAR_OUTPUT
  BAJARCUCHILLA : BOOL ;
  EXPULSARPLANCHA : BOOL ;
  bit_ok : BOOL ;
  STBY : BOOL ;
END_VAR
VAR_TEMP
  x51 : BOOL ;
  x52 : BOOL ;
  x53 : BOOL ;
  s3 : BOOL ;
  FP_BDT : BOOL ;
  X50 : BOOL ;
  FP_START : BOOL ;
END_VAR
BEGIN
NETWORK
TITLE = Arranque
      A     #bit_de_trabajo;
      FP    #FP_BDT;
      S     #X50;
      R     #x51;
      R     #x52;
      R     #x53;
      R     #s3;
NETWORK
TITLE = de x51 a x52
      A     #x51;
      A     #SENSORABAJO;
      R     #x51;
      S     #x52;
NETWORK
TITLE = de x52 a x53
      A     #x52;
      A     #SENSORARRIBA;
      R     #x52;
      S     #x53;
NETWORK
TITLE = de x53 a s3
      A     #x53;
      A     #EXPULSADA;
      R     #x53;
      S     #s3;
NETWORK
TITLE = Accion x51
      A     #x51;
      =     #BAJARCUCHILLA;
NETWORK
TITLE = Accion x53
      A     #x53;
      =     #EXPULSARPLANCHA;
NETWORK
TITLE = Accion final
      A     #s3;
      =     #bit_ok;
NETWORK
TITLE =
      A     #s3;
      A     #OK;
      R     #s3;
      S     #X50;
NETWORK
TITLE =
      A     #X50;
      A     #START;
      FP    #FP_START;
      R     #X50;
      S     #x51;
NETWORK
TITLE =
      A     #X50;
      =     #STBY;
END_FUNCTION

FUNCTION "PESAJE" : VOID	// FC 2
TITLE = PESAJE
VERSION : 0.1
VAR_INPUT
  in : INT ;
  PESO_SARTEN : REAL ;
  PESO_CACEROLA : REAL ;
  PESO_WOK : REAL ;
  PESO_PAELLERA : REAL ;
  bit_de_trabajo : BOOL ;
  RECIBIDO : BOOL ;
  START : BOOL ;
END_VAR
VAR_OUTPUT
  stby : BOOL ;
  SARTEN : BOOL ;
  CACEROLA : BOOL ;
  WOK : BOOL ;
  PAELLERA : BOOL ;
  PESO_OUT : REAL ;
END_VAR
VAR_TEMP
  retFC105 : WORD ;
  x121 : BOOL ;
  x122 : BOOL ;
  x123 : BOOL ;
  x124 : BOOL ;
  m3 : BOOL ;
  x120 : BOOL ;
  FP_BDT : BOOL ;
  FP_START : BOOL ;
  PESO : REAL ;
END_VAR
BEGIN
NETWORK
TITLE = Pesado
      A     #m3;
      CALL  "SCALE" (
           $1                       := #in,
           $2                       := L#1133903872,
           $3                       := L#0,
           $4                       := FALSE,
           $5                       := #retFC105,
           $6                       := #PESO);
NETWORK
TITLE =
      A     #x120;
      A     #START;
      FP    #FP_START;
      R     #x120;
      S     #m3;
NETWORK
TITLE = Arranque
      A     #bit_de_trabajo;
      FP    #FP_BDT;
      S     #x120;
      R     #m3;
      R     #x121;
      R     #x122;
      R     #x123;
      R     #x124;
NETWORK
TITLE =
      A(;
      L     #PESO_SARTEN;
      L     5.000000e+00;
      +R;
      L     #PESO;
      >R;
      );
      A(;
      L     #PESO_SARTEN;
      L     5.000000e+00;
      -R;
      L     #PESO;
      <R;
      );
      A     #m3;
      R     #m3;
      S     #x121;
NETWORK
TITLE =
      L     #PESO;
      T     #PESO_OUT;
NETWORK
TITLE =
      A(;
      L     #PESO_CACEROLA;
      L     5.000000e+00;
      +R;
      L     #PESO;
      >R;
      );
      A(;
      L     #PESO_CACEROLA;
      L     5.000000e+00;
      -R;
      L     #PESO;
      <R;
      );
      A     #m3;
      R     #m3;
      S     #x122;
NETWORK
TITLE =
      A(;
      L     #PESO_WOK;
      L     5.000000e+00;
      +R;
      L     #PESO;
      >R;
      );
      A(;
      L     #PESO_WOK;
      L     5.000000e+00;
      -R;
      L     #PESO;
      <R;
      );
      A     #m3;
      R     #m3;
      S     #x123;
NETWORK
TITLE =
      A(;
      L     #PESO_PAELLERA;
      L     5.000000e+00;
      +R;
      L     #PESO;
      >R;
      );
      A(;
      L     #PESO_PAELLERA;
      L     5.000000e+00;
      -R;
      L     #PESO;
      <R;
      );
      A     #m3;
      R     #m3;
      S     #x124;
NETWORK
TITLE = TRATAMIENTO SALIDAS
      A     #x121;
      =     #SARTEN;
      A     #x122;
      =     #CACEROLA;
      A     #x123;
      =     #WOK;
      A     #x124;
      =     #PAELLERA;
      A     #x120;
      =     #stby;
NETWORK
TITLE = Paso de estado pesado a stby
      A(;
      A     #x121;
      O     #x122;
      O     #x123;
      O     #x124;
      );
      A     #RECIBIDO;
      R     #x121;
      R     #x122;
      R     #x123;
      R     #x124;
      S     #x120;
END_FUNCTION

// FC 105: know-how protected block, not included

DATA_BLOCK "Global"	// DB 1
VERSION : 0.1
  STRUCT
   PESO_CACEROLA : REAL  := 1.000000e+002;	//Peso Bobina Cacerolas
   PESO_WOK : REAL  := 1.100000e+002;	//Peso Bobina Wok
   PESO_SARTEN : REAL  := 1.200000e+002;	//Peso Bobina Sarten
   PESO_PAELLERA : REAL  := 1.300000e+002;	//Peso Bobina Paellera
   PLANCHAS : WORD  := W#16#100;	//Número de planchas por bobina
  END_STRUCT ;	
BEGIN
   PESO_CACEROLA := 1.000000e+02;
   PESO_WOK := 1.100000e+02;
   PESO_SARTEN := 1.200000e+02;
   PESO_PAELLERA := 1.300000e+02;
   PLANCHAS := W#16#100;
END_DATA_BLOCK

DATA_BLOCK "INFO_BOB"	// DB 4
VERSION : 0.1
  STRUCT
   CENTRO_CACEROLA : INT  := 10;	//Variable provisional
   CENTRO_SARTEN : INT  := 20;
   CENTRO_WOK : INT  := 30;
   CENTRO_PAELLERA : INT  := 40;
  END_STRUCT ;	
BEGIN
END_DATA_BLOCK

DATA_BLOCK DB 5
VERSION : 0.0
"MULT_GEN"
BEGIN
END_DATA_BLOCK

ORGANIZATION_BLOCK "Cycle Execution"	// OB 1
TITLE = "Main Program Sweep (Cycle)"
VERSION : 0.1
VAR_TEMP
  OB1_EV_CLASS : BYTE ;	//Bits 0-3 = 1 (Coming event), Bits 4-7 = 1 (Event class 1)
  OB1_SCAN_1 : BYTE ;	//1 (Cold restart scan 1 of OB 1), 3 (Scan 2-n of OB 1)
  OB1_PRIORITY : BYTE ;	//Priority of OB Execution
  OB1_OB_NUMBR : BYTE ;	//1 (Organization block 1, OB1)
  OB1_RESERVED_1 : BYTE ;	//Reserved for system
  OB1_RESERVED_2 : BYTE ;	//Reserved for system
  OB1_PREV_CYCLE : INT ;	//Cycle time of previous OB1 scan (milliseconds)
  OB1_MIN_CYCLE : INT ;	//Minimum cycle time of OB1 (milliseconds)
  OB1_MAX_CYCLE : INT ;	//Maximum cycle time of OB1 (milliseconds)
  OB1_DATE_TIME : DATE_AND_TIME ;	//Date and time OB1 started
END_VAR
BEGIN
NETWORK
TITLE =
      SET;
      CALL  "MULT_GEN" , DB 5 (
           START                    := "START",
           BIT_DE_TRABAJO           := "BIT_DE_TRABAJO",
           BOBINA_COLOCADA          := "BOBINA_COLOCADA",
           MCENTRO                  := "MCENTRO",
           IN_PESAJE                := "IN_PESAJE",
           S_SARTEN                 := "S_SARTEN",
           S_CACEROLA               := "S_CACEROLA",
           S_WOK                    := "S_WOK",
           S_PAELLERA               := "S_PAELLERA",
           PRESENCIA                := "PRESENCIA",
           CONTADOR                 := "CONTADOR",
           PALET                    := "PALET",
           SENSORARRIBA             := "SENSORARRIBA",
           SENSORABAJO              := "SENSORABAJO",
           EXPULSADA                := "EXPULSADA",
           PESO_OUT                 := "PESO_OUT",
           ABRIRMCENTRO             := "ABRIRMCENTRO",
           CERRARMCENTRO            := "DESBOBINAR",
           DESBOBINAR               := "EXPULSAR_BOBINA",
           EXPULSAR_BOBINA          := "PRENSA",
           PRENSA                   := "EXPULSAR_PLANCHA",
           EXPULSAR_PLANCHA         := "BAJAR_CUCHILLA",
           BAJAR_CUCHILLA           := Q 100.7,
           EXPULSAR_PALET           := "EXPULSAR_PALET",
           STBY                     := "STBY");
END_ORGANIZATION_BLOCK
